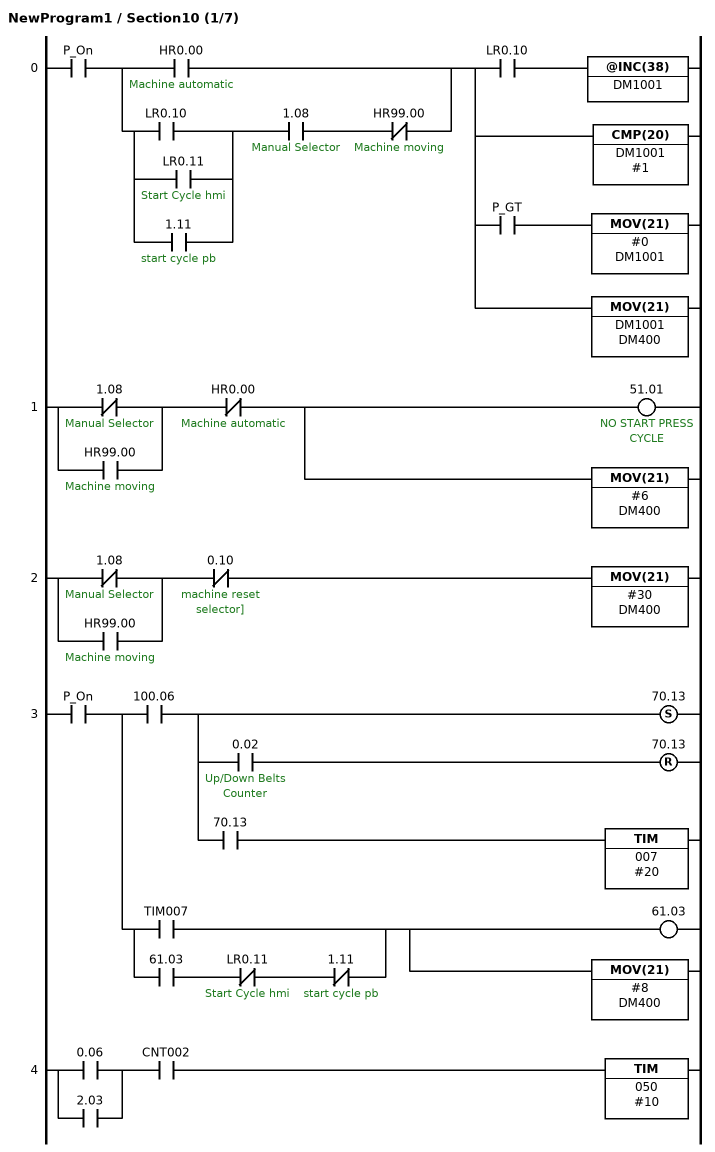
; [picture p48: NewProgram1 / Section10, rungs 0-4]
; rung 0
LD P_On
LD HR0.00  ; Machine automatic
LD LR0.10
OR LR0.11  ; Start Cycle hmi
OR 1.11  ; start cycle pb
AND 1.08  ; Manual Selector
ANDNOT HR99.00  ; Machine moving
ORLD
ANDLD
OUT TR0
AND LR0.10
@INC(38) DM1001
LD TR0
CMP(20) DM1001 #1
AND P_GT
MOV(21) #0 DM1001
LD TR0
MOV(21) DM1001 DM400
; rung 1
LDNOT 1.08  ; Manual Selector
OR HR99.00  ; Machine moving
ANDNOT HR0.00  ; Machine automatic
OUT 51.01  ; NO START PRESS CYCLE
MOV(21) #6 DM400
; rung 2
LDNOT 1.08  ; Manual Selector
OR HR99.00  ; Machine moving
ANDNOT 0.10  ; machine reset selector]
MOV(21) #30 DM400
; rung 3
LD P_On
OUT TR0
AND 100.06
OUT TR1
SET 70.13
AND 0.02  ; Up/Down Belts Counter
RSET 70.13
LD TR1
AND 70.13
TIM 007 #20
LD TR0
LD TIM007
LD 61.03
ANDNOT LR0.11  ; Start Cycle hmi
ANDNOT 1.11  ; start cycle pb
ORLD
ANDLD
OUT 61.03
MOV(21) #8 DM400
; rung 4
LD 0.06
OR 2.03
AND CNT002
TIM 050 #10

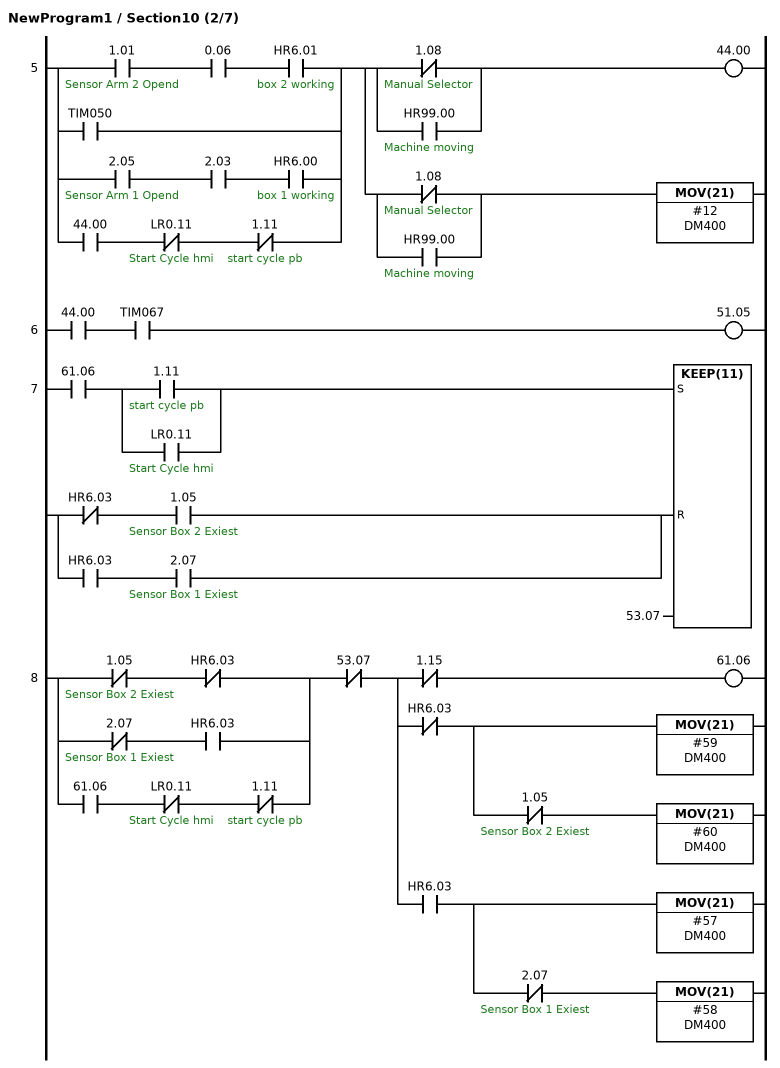
; rung 5
LD 1.01  ; Sensor Arm 2 Opend
AND 0.06
AND HR6.01  ; box 2 working
OR TIM050
LD 2.05  ; Sensor Arm 1 Opend
AND 2.03
AND HR6.00  ; box 1 working
ORLD
LD 44.00
ANDNOT LR0.11  ; Start Cycle hmi
ANDNOT 1.11  ; start cycle pb
ORLD
OUT TR0
LDNOT 1.08  ; Manual Selector
OR HR99.00  ; Machine moving
ANDLD
OUT 44.00
LD TR0
LDNOT 1.08  ; Manual Selector
OR HR99.00  ; Machine moving
ANDLD
MOV(21) #12 DM400
; rung 6
LD 44.00
AND TIM067
OUT 51.05
; rung 7
LD 61.06
LD 1.11  ; start cycle pb
OR LR0.11  ; Start Cycle hmi
ANDLD
LDNOT HR6.03
AND 1.05  ; Sensor Box 2 Exiest
LD HR6.03
AND 2.07  ; Sensor Box 1 Exiest
ORLD
KEEP(11) 53.07
; rung 8
LDNOT 1.05  ; Sensor Box 2 Exiest
ANDNOT HR6.03
LDNOT 2.07  ; Sensor Box 1 Exiest
AND HR6.03
ORLD
LD 61.06
ANDNOT LR0.11  ; Start Cycle hmi
ANDNOT 1.11  ; start cycle pb
ORLD
ANDNOT 53.07
OUT TR0
ANDNOT 1.15
OUT 61.06
LD TR0
ANDNOT HR6.03
MOV(21) #59 DM400
ANDNOT 1.05  ; Sensor Box 2 Exiest
MOV(21) #60 DM400
LD TR0
AND HR6.03
MOV(21) #57 DM400
ANDNOT 2.07  ; Sensor Box 1 Exiest
MOV(21) #58 DM400

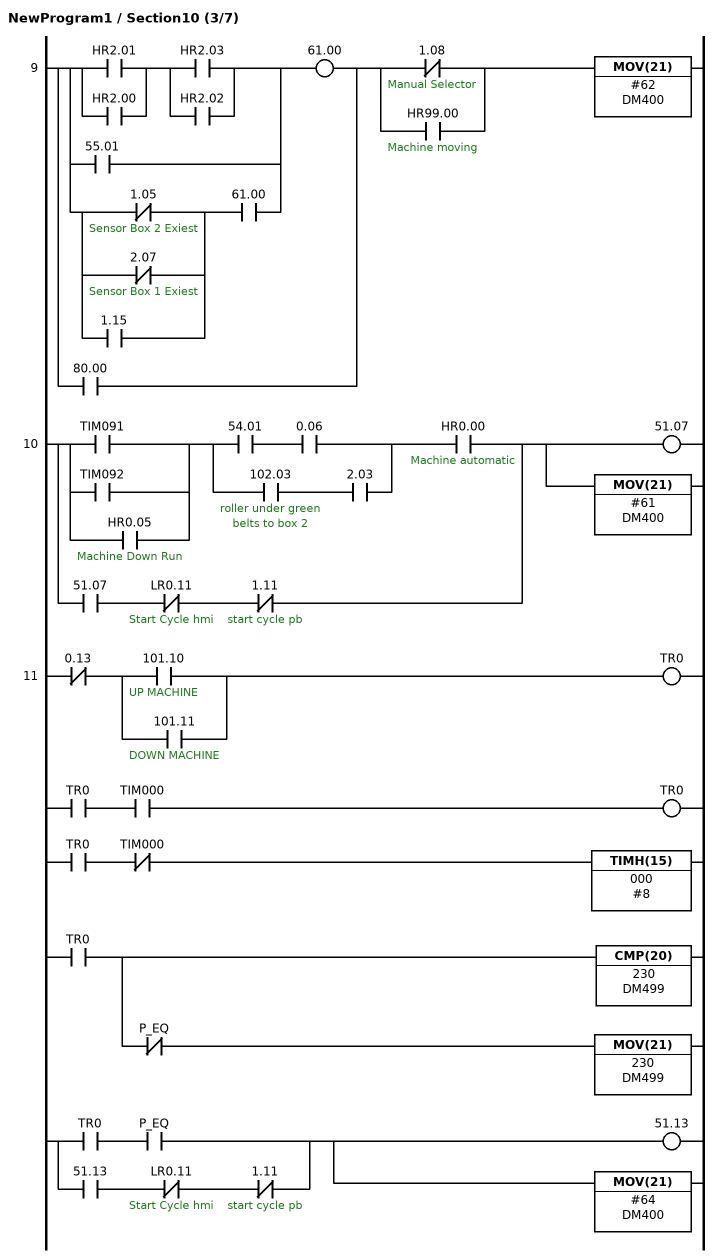
; rung 9
LD HR2.01
OR HR2.00
LD HR2.03
OR HR2.02
ANDLD
OR 55.01
LDNOT 1.05  ; Sensor Box 2 Exiest
ORNOT 2.07  ; Sensor Box 1 Exiest
OR 1.15
AND 61.00
ORLD
OUT 61.00
OR 80.00
LDNOT 1.08  ; Manual Selector
OR HR99.00  ; Machine moving
ANDLD
MOV(21) #62 DM400
; rung 10
LD TIM091
OR TIM092
OR HR0.05  ; Machine Down Run
LD 54.01
AND 0.06
LD 102.03  ; roller under green belts to box 2
AND 2.03
ORLD
ANDLD
AND HR0.00  ; Machine automatic
LD 51.07
ANDNOT LR0.11  ; Start Cycle hmi
ANDNOT 1.11  ; start cycle pb
ORLD
OUT 51.07
MOV(21) #61 DM400
; rung 11
LDNOT 0.13
LD 101.10  ; UP MACHINE
OR 101.11  ; DOWN MACHINE
ANDLD
OUT TR0
ANDNOT TIM000
TIMH(15) 000 #8
LD TR0
AND TIM000
OUT TR0
CMP(20) 230 DM499
ANDNOT P_EQ
MOV(21) 230 DM499
LD TR0
AND P_EQ
LD 51.13
ANDNOT LR0.11  ; Start Cycle hmi
ANDNOT 1.11  ; start cycle pb
ORLD
OUT 51.13
MOV(21) #64 DM400

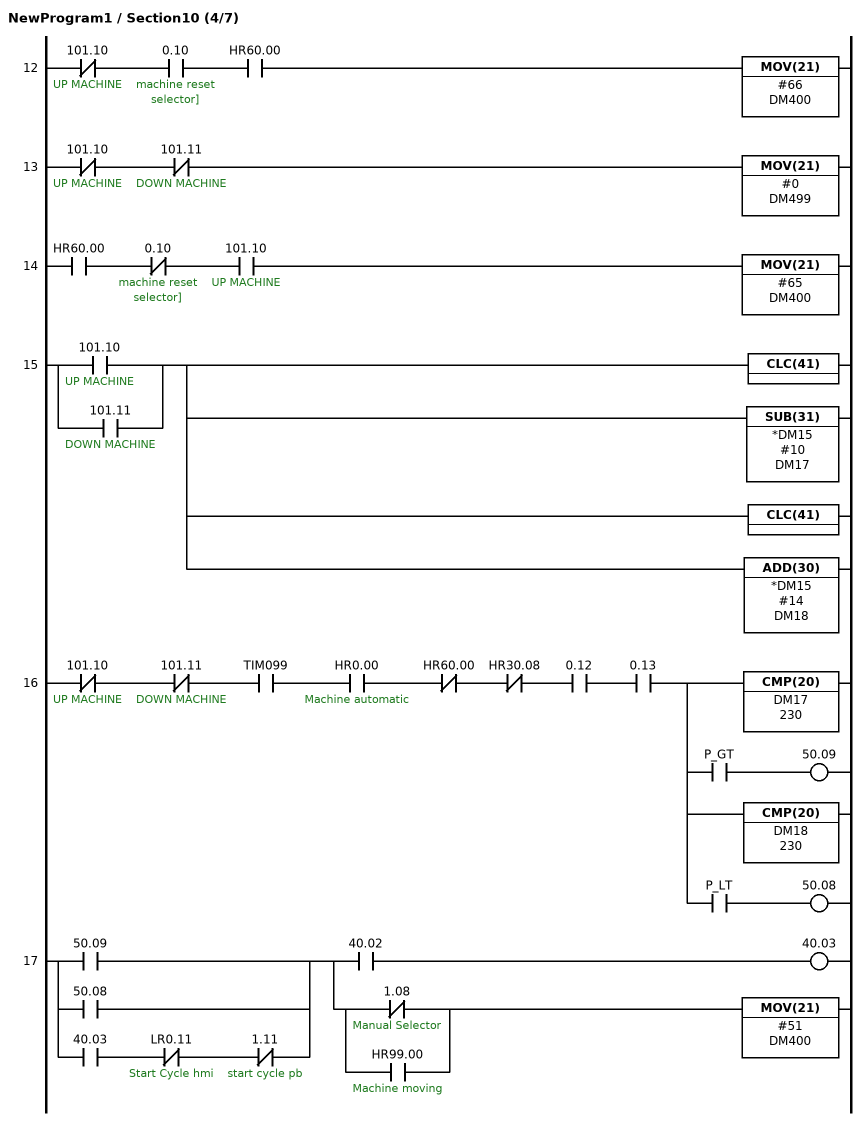
; rung 12
LDNOT 101.10  ; UP MACHINE
AND 0.10  ; machine reset selector]
AND HR60.00
MOV(21) #66 DM400
; rung 13
LDNOT 101.10  ; UP MACHINE
ANDNOT 101.11  ; DOWN MACHINE
MOV(21) #0 DM499
; rung 14
LD HR60.00
ANDNOT 0.10  ; machine reset selector]
AND 101.10  ; UP MACHINE
MOV(21) #65 DM400
; rung 15
LD 101.10  ; UP MACHINE
OR 101.11  ; DOWN MACHINE
CLC(41)
SUB(31) *DM15 #10 DM17
CLC(41)
ADD(30) *DM15 #14 DM18
; rung 16
LDNOT 101.10  ; UP MACHINE
ANDNOT 101.11  ; DOWN MACHINE
AND TIM099
AND HR0.00  ; Machine automatic
ANDNOT HR60.00
ANDNOT HR30.08
AND 0.12
AND 0.13
OUT TR0
CMP(20) DM17 230
AND P_GT
OUT 50.09
LD TR0
CMP(20) DM18 230
AND P_LT
OUT 50.08
; rung 17
LD 50.09
OR 50.08
LD 40.03
ANDNOT LR0.11  ; Start Cycle hmi
ANDNOT 1.11  ; start cycle pb
ORLD
OUT TR0
AND 40.02
OUT 40.03
LD TR0
LDNOT 1.08  ; Manual Selector
OR HR99.00  ; Machine moving
ANDLD
MOV(21) #51 DM400

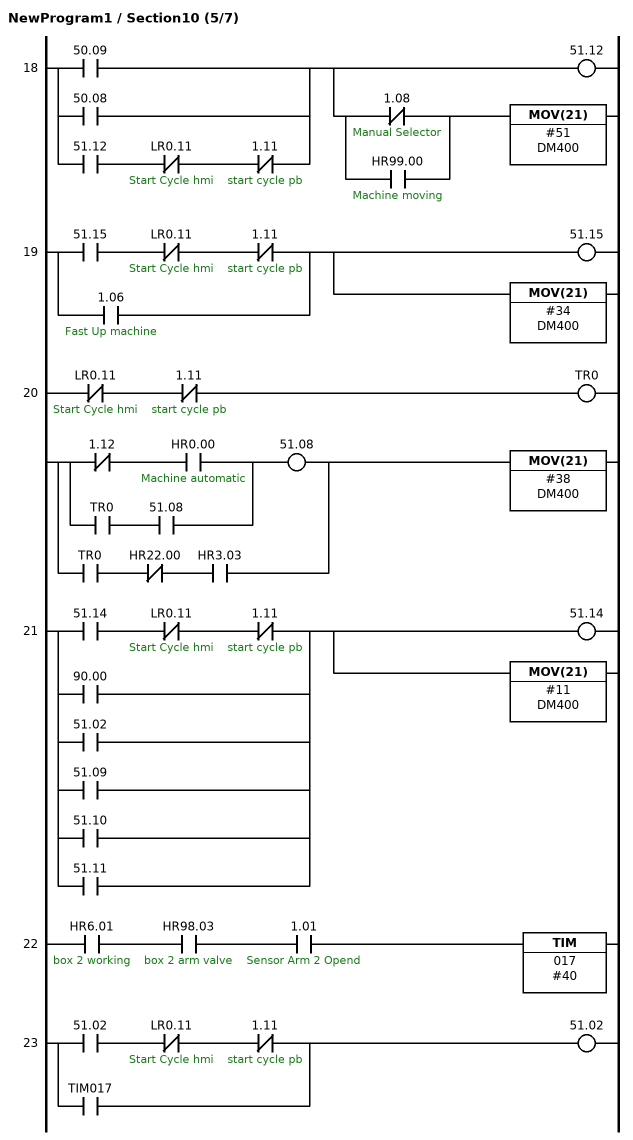
; rung 18
LD 50.09
OR 50.08
LD 51.12
ANDNOT LR0.11  ; Start Cycle hmi
ANDNOT 1.11  ; start cycle pb
ORLD
OUT 51.12
LDNOT 1.08  ; Manual Selector
OR HR99.00  ; Machine moving
ANDLD
MOV(21) #51 DM400
; rung 19
LD 51.15
ANDNOT LR0.11  ; Start Cycle hmi
ANDNOT 1.11  ; start cycle pb
OR 1.06  ; Fast Up machine
OUT 51.15
MOV(21) #34 DM400
; rung 20
LDNOT 1.12
AND HR0.00  ; Machine automatic
LDNOT LR0.11  ; Start Cycle hmi
ANDNOT 1.11  ; start cycle pb
OUT TR0
AND 51.08
ORLD
OUT 51.08
LD TR0
ANDNOT HR22.00
AND HR3.03
ORLD
MOV(21) #38 DM400
; rung 21
LD 51.14
ANDNOT LR0.11  ; Start Cycle hmi
ANDNOT 1.11  ; start cycle pb
OR 90.00
OR 51.02
OR 51.09
OR 51.10
OR 51.11
OUT 51.14
MOV(21) #11 DM400
; rung 22
LD HR6.01  ; box 2 working
AND HR98.03  ; box 2 arm valve
AND 1.01  ; Sensor Arm 2 Opend
TIM 017 #40
; rung 23
LD 51.02
ANDNOT LR0.11  ; Start Cycle hmi
ANDNOT 1.11  ; start cycle pb
OR TIM017
OUT 51.02

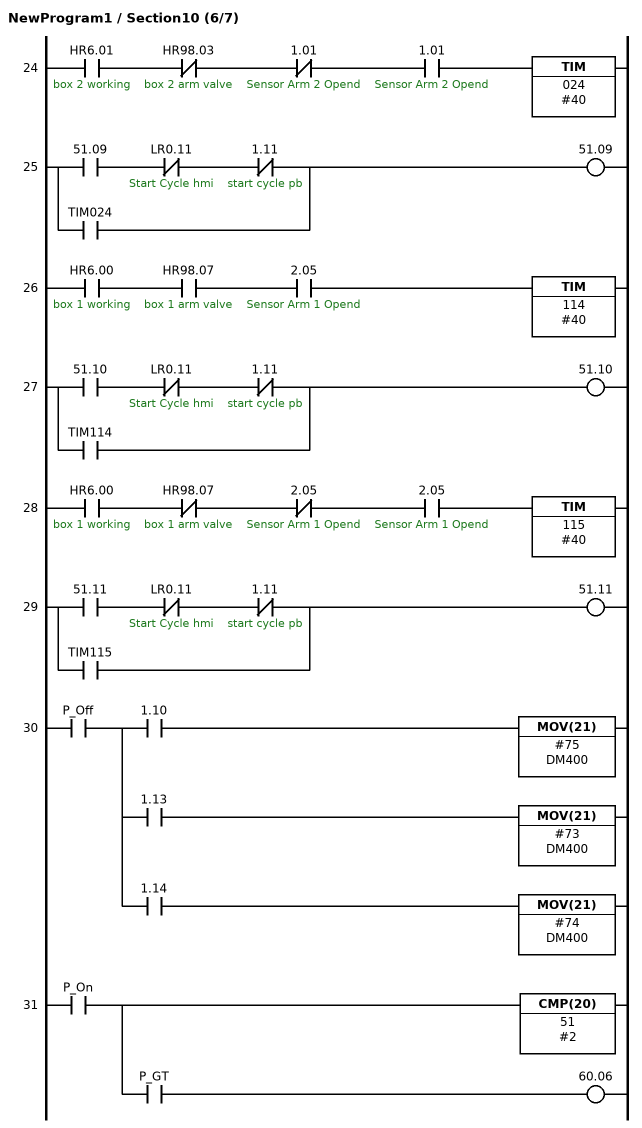
; rung 24
LD HR6.01  ; box 2 working
ANDNOT HR98.03  ; box 2 arm valve
ANDNOT 1.01  ; Sensor Arm 2 Opend
AND 1.01  ; Sensor Arm 2 Opend
TIM 024 #40
; rung 25
LD 51.09
ANDNOT LR0.11  ; Start Cycle hmi
ANDNOT 1.11  ; start cycle pb
OR TIM024
OUT 51.09
; rung 26
LD HR6.00  ; box 1 working
AND HR98.07  ; box 1 arm valve
AND 2.05  ; Sensor Arm 1 Opend
TIM 114 #40
; rung 27
LD 51.10
ANDNOT LR0.11  ; Start Cycle hmi
ANDNOT 1.11  ; start cycle pb
OR TIM114
OUT 51.10
; rung 28
LD HR6.00  ; box 1 working
ANDNOT HR98.07  ; box 1 arm valve
ANDNOT 2.05  ; Sensor Arm 1 Opend
AND 2.05  ; Sensor Arm 1 Opend
TIM 115 #40
; rung 29
LD 51.11
ANDNOT LR0.11  ; Start Cycle hmi
ANDNOT 1.11  ; start cycle pb
OR TIM115
OUT 51.11
; rung 30
LD P_Off
OUT TR0
AND 1.10
MOV(21) #75 DM400
LD TR0
AND 1.13
MOV(21) #73 DM400
LD TR0
AND 1.14
MOV(21) #74 DM400
; rung 31
LD P_On
CMP(20) 51 #2
AND P_GT
OUT 60.06

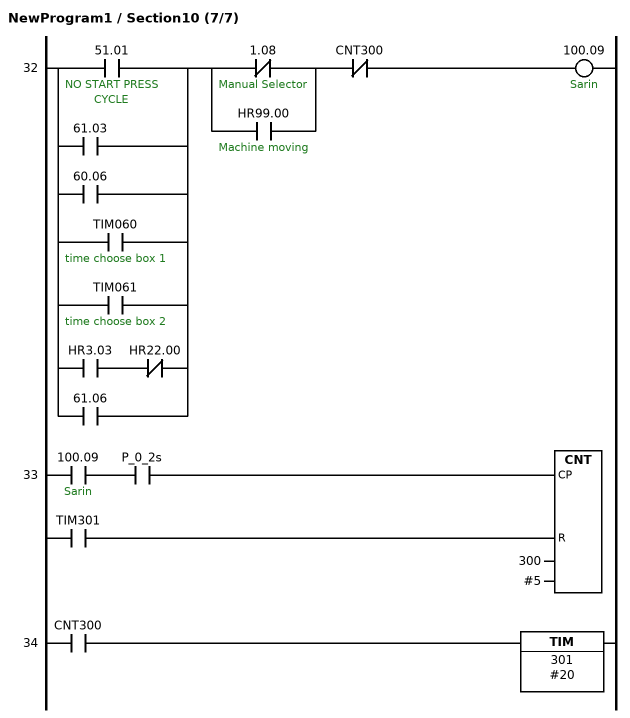
; rung 32
LD 51.01  ; NO START PRESS CYCLE
OR 61.03
OR 60.06
OR TIM060  ; time choose box 1
OR TIM061  ; time choose box 2
LD HR3.03
ANDNOT HR22.00
ORLD
OR 61.06
LDNOT 1.08  ; Manual Selector
OR HR99.00  ; Machine moving
ANDLD
ANDNOT CNT300
OUT 100.09  ; Sarin
; rung 33
LD 100.09  ; Sarin
AND P_0_2s
LD TIM301
CNT 300 #5
; rung 34
LD CNT300
TIM 301 #20

### Section Section11

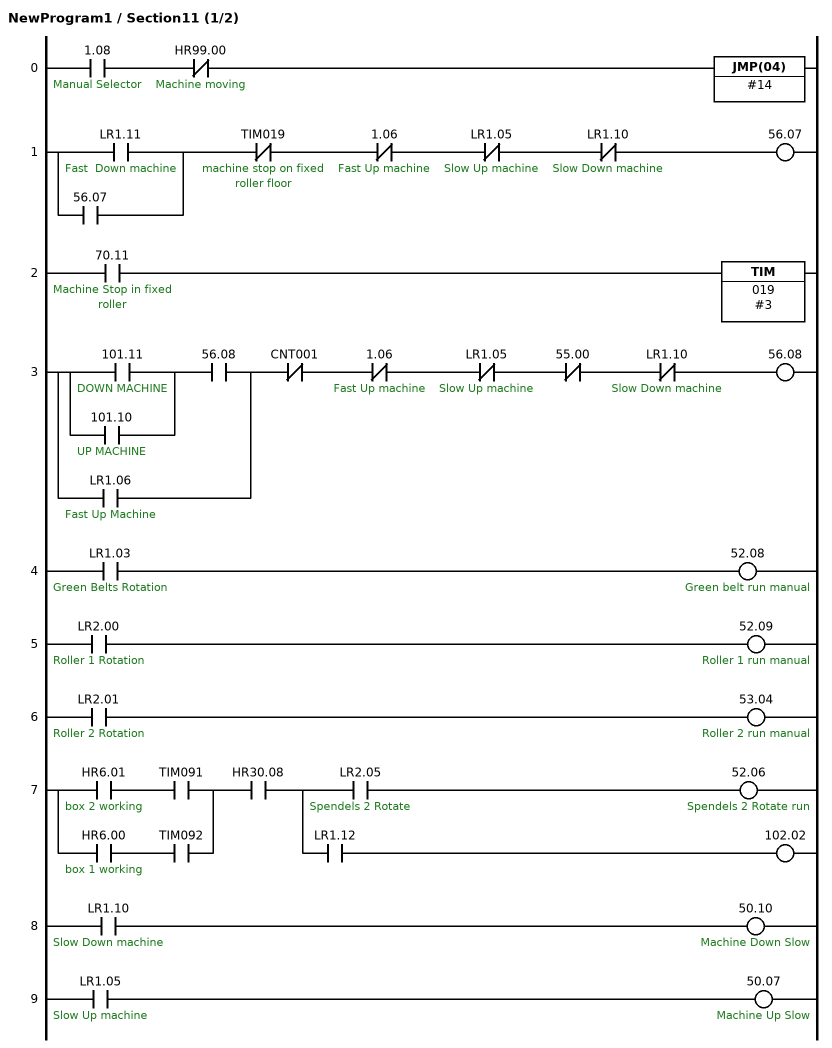
; rung 0
LD 1.08  ; Manual Selector
ANDNOT HR99.00  ; Machine moving
JMP(04) #14
; rung 1
LD LR1.11  ; Fast  Down machine
OR 56.07
ANDNOT TIM019  ; machine stop on fixed roller floor
ANDNOT 1.06  ; Fast Up machine
ANDNOT LR1.05  ; Slow Up machine
ANDNOT LR1.10  ; Slow Down machine
OUT 56.07
; rung 2
LD 70.11  ; Machine Stop in fixed roller
TIM 019 #3
; rung 3
LD 101.11  ; DOWN MACHINE
OR 101.10  ; UP MACHINE
AND 56.08
OR LR1.06  ; Fast Up Machine
ANDNOT CNT001
ANDNOT 1.06  ; Fast Up machine
ANDNOT LR1.05  ; Slow Up machine
ANDNOT 55.00
ANDNOT LR1.10  ; Slow Down machine
OUT 56.08
; rung 4
LD LR1.03  ; Green Belts Rotation
OUT 52.08  ; Green belt run manual
; rung 5
LD LR2.00  ; Roller 1 Rotation
OUT 52.09  ; Roller 1 run manual
; rung 6
LD LR2.01  ; Roller 2 Rotation
OUT 53.04  ; Roller 2 run manual
; rung 7
LD HR6.01  ; box 2 working
AND TIM091
LD HR6.00  ; box 1 working
AND TIM092
ORLD
AND HR30.08
OUT TR0
AND LR2.05  ; Spendels 2 Rotate
OUT 52.06  ; Spendels 2 Rotate run
LD TR0
AND LR1.12
OUT 102.02
; rung 8
LD LR1.10  ; Slow Down machine
OUT 50.10  ; Machine Down Slow
; rung 9
LD LR1.05  ; Slow Up machine
OUT 50.07  ; Machine Up Slow

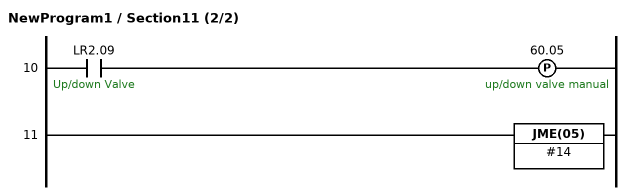
; rung 10
LD LR2.09  ; Up/down Valve
DIFU(13) 60.05  ; up/down valve manual
; rung 11
JME(05) #14

### Section Section12

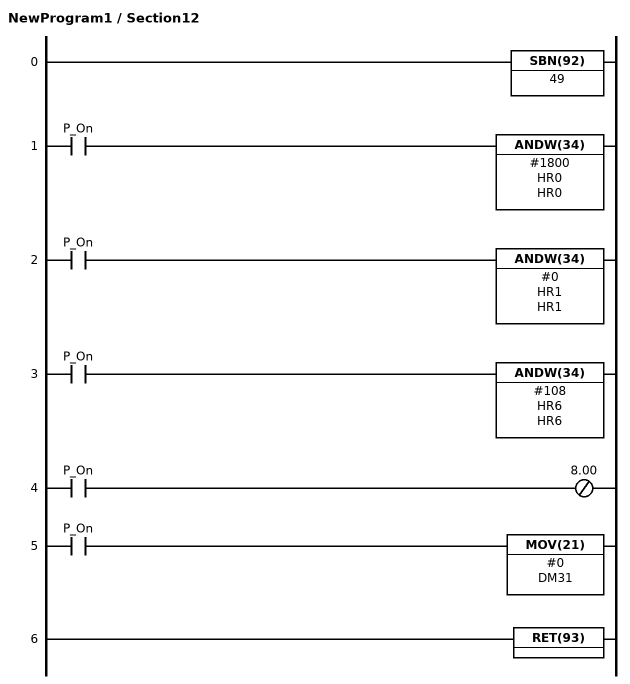
; rung 0
SBN(92) 49
; rung 1
LD P_On
ANDW(34) #1800 HR0 HR0
; rung 2
LD P_On
ANDW(34) #0 HR1 HR1
; rung 3
LD P_On
ANDW(34) #108 HR6 HR6
; rung 4
LD P_On
OUTNOT 8.00
; rung 5
LD P_On
MOV(21) #0 DM31
; rung 6
RET(93)

### Section Section13

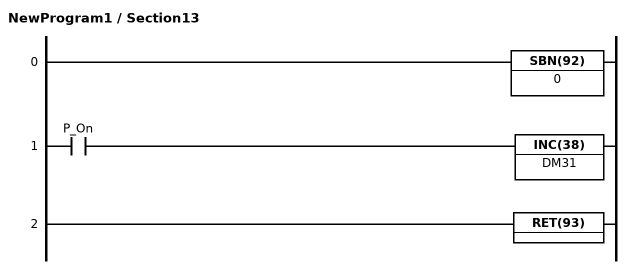
; rung 0
SBN(92) 0
; rung 1
LD P_On
INC(38) DM31
; rung 2
RET(93)

### Section Section14
; rung 0
END(01)

### Section Section15

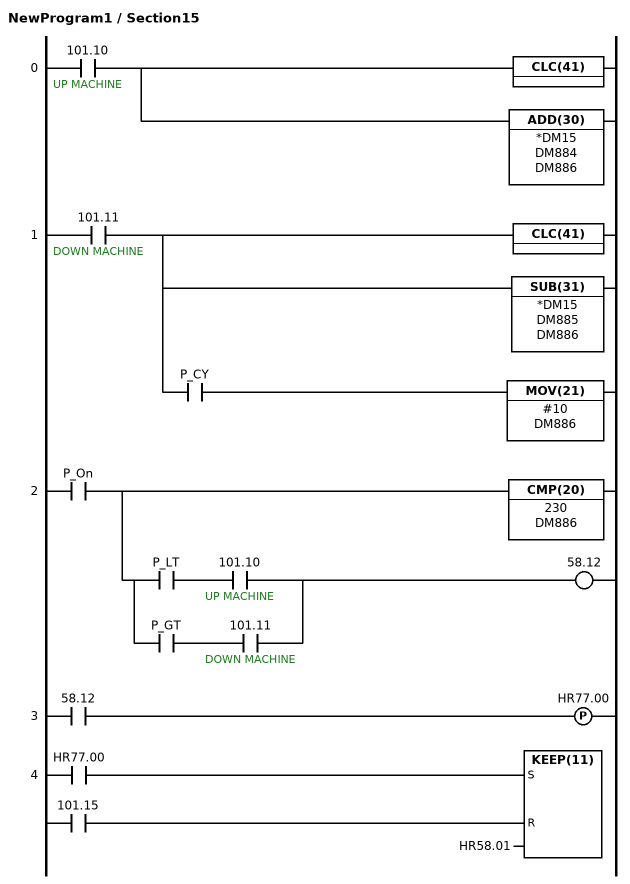
; rung 0
LD 101.10  ; UP MACHINE
CLC(41)
ADD(30) *DM15 DM884 DM886
; rung 1
LD 101.11  ; DOWN MACHINE
CLC(41)
SUB(31) *DM15 DM885 DM886
AND P_CY
MOV(21) #10 DM886
; rung 2
LD P_On
CMP(20) 230 DM886
LD P_LT
AND 101.10  ; UP MACHINE
LD P_GT
AND 101.11  ; DOWN MACHINE
ORLD
ANDLD
OUT 58.12
; rung 3
LD 58.12
DIFU(13) HR77.00
; rung 4
LD HR77.00
LD 101.15
KEEP(11) HR58.01
; rung 5
END(01)